// TwinCAT 3 PLC project FiniteStateMachine
// ProgramVersion: 3.1.4023.0
// libraries:
//   Tc2_Standard, * (Beckhoff Automation GmbH)
//   Tc2_System, * (Beckhoff Automation GmbH)
//   Tc3_Module, * (Beckhoff Automation GmbH)
// project tree:
//   / PlcTask.TcTTO
//   POUs/ MAIN.TcPOU, Prg_FSM.TcPOU
// real-time tasks:
//   TASK PlcTask: cycle T#10ms, priority 20, ADS port 350

CONFIGURATION FiniteStateMachine
    RESOURCE PLC ON TwinCAT3
        TASK PlcTask(INTERVAL := T#10ms, PRIORITY := 20);
        PROGRAM MAIN WITH PlcTask : MAIN;
    END_RESOURCE
END_CONFIGURATION

// ---- POUs/MAIN.TcPOU
PROGRAM MAIN
VAR
END_VAR

Prg_FSM();

END_PROGRAM

// ---- POUs/Prg_FSM.TcPOU
PROGRAM Prg_FSM
VAR
	Start: BOOL;
	Stop: BOOL;
	Mixer: BOOL;
	Pump: BOOL;
	Gate: BOOL;
	Timer1: TON;
	State: INT;
	StartT: R_TRIG;
	StopT: R_TRIG;
END_VAR


StartT(CLK:=Start);
StopT(CLK:=Stop);

CASE State OF
	0:
		IF StartT.Q THEN
			State:=1;
		ELSE
			State:=0;
		END_IF
	
	1:
		Mixer:=TRUE;
		Timer1(IN:=TRUE, PT:=T#5S, ET=>);
		IF Timer1.Q THEN
			Timer1(IN:=FALSE);
			State:=2;
		END_IF
	2:
		Pump:=TRUE;
		Timer1(IN:=TRUE, PT:=T#5S, ET=>);
		IF Timer1.Q THEN
			Timer1(IN:=FALSE);
			pump:=FALSE;
			State:=3;
		ELSE
			State:=2;
		END_IF
	3:
		Timer1(IN:=TRUE, PT:=T#5S, ET=>);
		IF Timer1.Q THEN
			Timer1(IN:=FALSE);
			Mixer:=FALSE;
			State:=4;
		ELSE
			State:=3;
		END_IF
	4:
		Gate:=TRUE;
		Timer1(IN:=TRUE, PT:=T#5S, ET=>);
		IF Timer1.Q THEN
			Timer1(IN:=FALSE);
			Gate:=FALSE;
			state:=0;
		ELSE
			State:=4;			
		END_IF
	
END_CASE

IF StopT.Q THEN
	State:=0;
	Mixer:=FALSE;
	Pump:=FALSE;
	Gate:=FALSE;
END_IF

END_PROGRAM
